// Mitsubishi GX Works2 project: inverter3   PLC: Q03UDV

PROGRAM MAIN
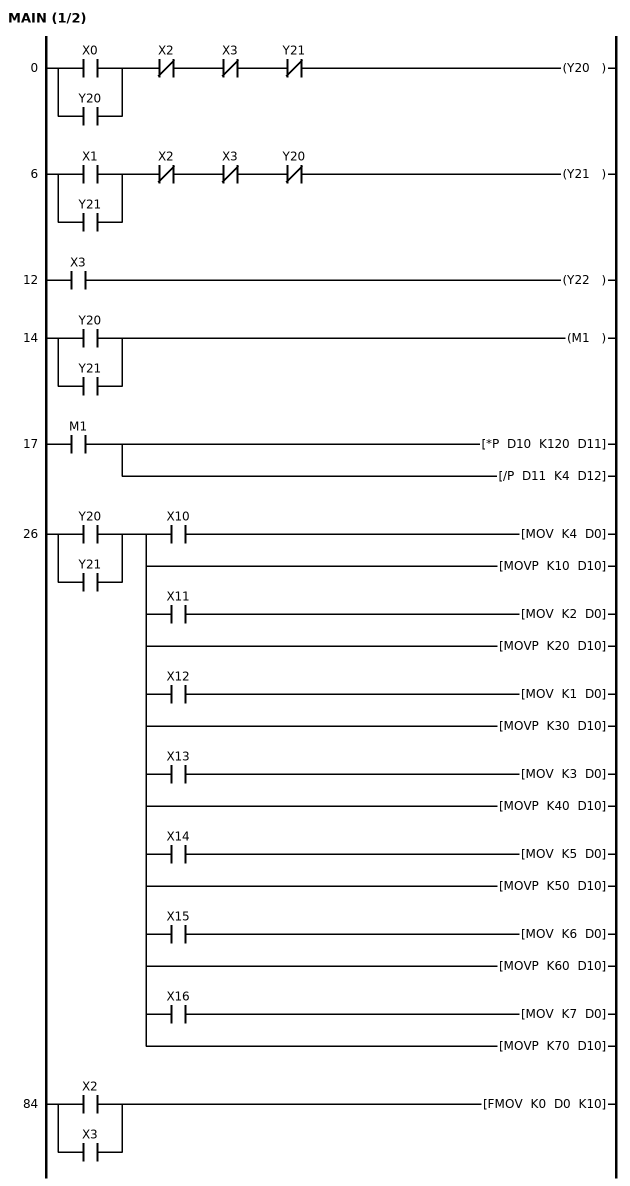
0     LD      X0
      OR      Y20
      ANI     X2
      ANI     X3
      ANI     Y21
      OUT     Y20
6     LD      X1
      OR      Y21
      ANI     X2
      ANI     X3
      ANI     Y20
      OUT     Y21
12    LD      X3
      OUT     Y22
14    LD      Y20
      OR      Y21
      OUT     M1
17    LD      M1
      *P      D10 K120 D11
      /P      D11 K4 D12
26    LD      Y20
      OR      Y21
      MPS
      AND     X10
      MOV     K4 D0
      MPP
      MOVP    K10 D10
      MPS
      AND     X11
      MOV     K2 D0
      MPP
      MOVP    K20 D10
      MPS
      AND     X12
      MOV     K1 D0
      MPP
      MOVP    K30 D10
      MPS
      AND     X13
      MOV     K3 D0
      MPP
      MOVP    K40 D10
      MPS
      AND     X14
      MOV     K5 D0
      MPP
      MOVP    K50 D10
      MPS
      AND     X15
      MOV     K6 D0
      MPP
      MOVP    K60 D10
      MPS
      AND     X16
      MOV     K7 D0
      MPP
      MOVP    K70 D10
84    LD      X2
      OR      X3
      FMOV    K0 D0 K10
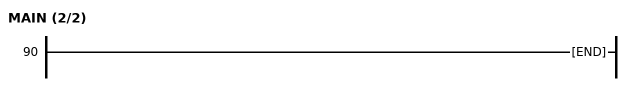
90    END
END_PROGRAM

PROGRAM MAIN1
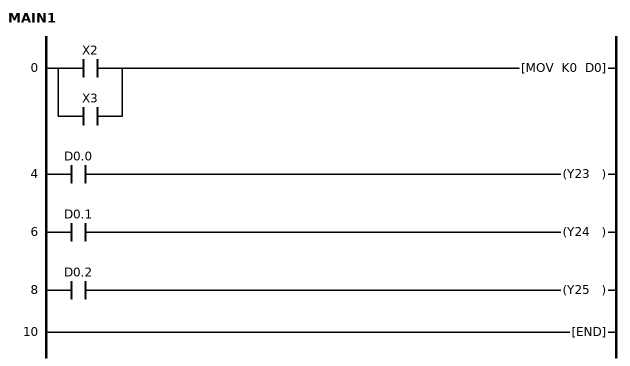
0     LD      X2
      OR      X3
      MOV     K0 D0
4     LD      D0.0
      OUT     Y23
6     LD      D0.1
      OUT     Y24
8     LD      D0.2
      OUT     Y25
10    END
END_PROGRAM
